// TIA Portal V18 export
FUNCTION "Function & start signal" : Void   // FC3, LAD
{ S7_Optimized_Access := 'TRUE' }
VERSION : 0.1
// stored: AutoNumber true, IsIECCheckEnabled false, SetENOAutomatically false, UDAEnableTagReadback false
   VAR_TEMP   // added for the SCL form of the ladder/FBD networks
      _w1 : Bool;
      _w2 : Bool;
      _w3 : Bool;
   END_VAR
BEGIN

REGION Network 1: Move dearing A Flowrate to Main register
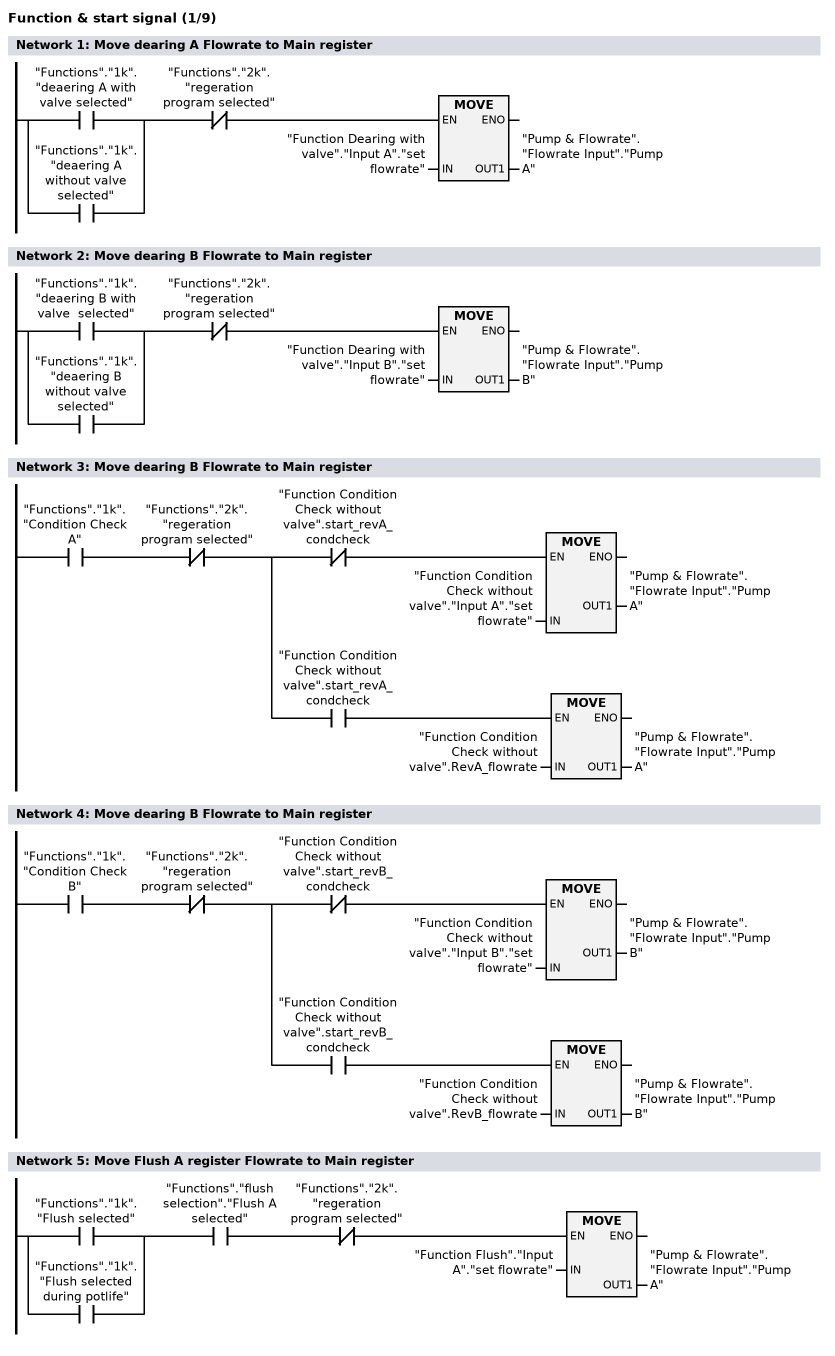
   IF ("Functions"."1k"."deaering A with valve selected" OR "Functions"."1k"."deaering A without valve selected") AND NOT "Functions"."2k"."regeration program selected" THEN
       "Pump & Flowrate"."Flowrate Input"."Pump A" := "Function Dearing with valve"."Input A"."set flowrate";
   END_IF;
END_REGION

REGION Network 2: Move dearing B Flowrate to Main register
   IF ("Functions"."1k"."deaering B with valve  selected" OR "Functions"."1k"."deaering B without valve  selected") AND NOT "Functions"."2k"."regeration program selected" THEN
       "Pump & Flowrate"."Flowrate Input"."Pump B" := "Function Dearing with valve"."Input B"."set flowrate";
   END_IF;
END_REGION

REGION Network 3: Move dearing B Flowrate to Main register
   #_w1 := "Functions"."1k"."Condition Check A" AND NOT "Functions"."2k"."regeration program selected";
   IF #_w1 AND NOT "Function ConditionCheck without valve".start_revA_condcheck THEN
       "Pump & Flowrate"."Flowrate Input"."Pump A" := "Function ConditionCheck without valve"."Input A"."set flowrate";
   END_IF;
   IF #_w1 AND "Function ConditionCheck without valve".start_revA_condcheck THEN
       "Pump & Flowrate"."Flowrate Input"."Pump A" := "Function ConditionCheck without valve".RevA_flowrate;
   END_IF;
END_REGION

REGION Network 4: Move dearing B Flowrate to Main register
   #_w1 := "Functions"."1k"."Condition Check B" AND NOT "Functions"."2k"."regeration program selected";
   IF #_w1 AND NOT "Function ConditionCheck without valve".start_revB_condcheck THEN
       "Pump & Flowrate"."Flowrate Input"."Pump B" := "Function ConditionCheck without valve"."Input B"."set flowrate";
   END_IF;
   IF #_w1 AND "Function ConditionCheck without valve".start_revB_condcheck THEN
       "Pump & Flowrate"."Flowrate Input"."Pump B" := "Function ConditionCheck without valve".RevB_flowrate;
   END_IF;
END_REGION

REGION Network 5: Move Flush A register Flowrate to Main register
   IF ("Functions"."1k"."Flush selected" OR "Functions"."1k"."Flush selected during potlife") AND "Functions"."flush selection"."Flush A selected" AND NOT "Functions"."2k"."regeration program selected" THEN
       "Pump & Flowrate"."Flowrate Input"."Pump A" := "Function Flush"."Input A"."set flowrate";
   END_IF;
END_REGION

REGION Network 6: Move Flush B register Flowrate to Main register
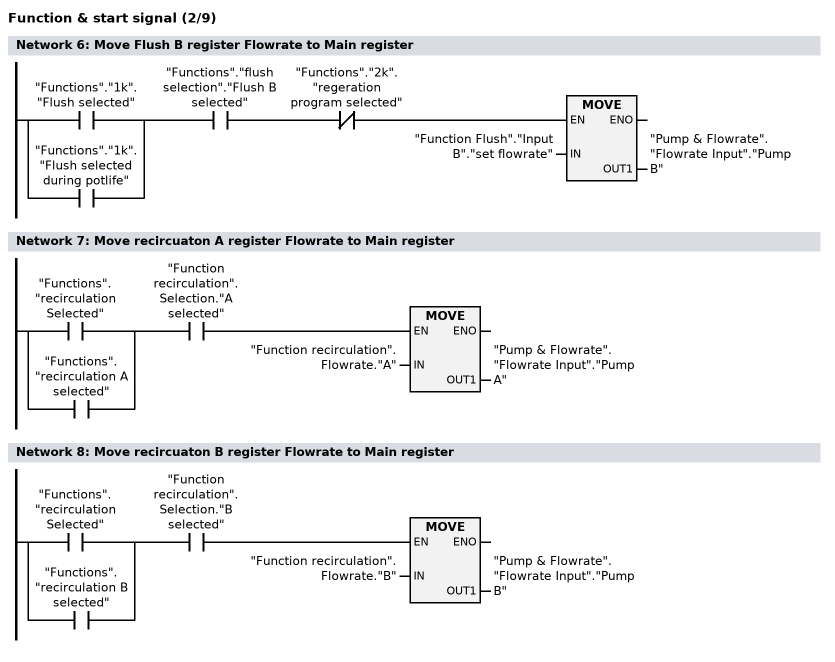
   IF ("Functions"."1k"."Flush selected" OR "Functions"."1k"."Flush selected during potlife") AND "Functions"."flush selection"."Flush B selected" AND NOT "Functions"."2k"."regeration program selected" THEN
       "Pump & Flowrate"."Flowrate Input"."Pump B" := "Function Flush"."Input B"."set flowrate";
   END_IF;
END_REGION

REGION Network 7: Move recircuaton A register Flowrate to Main register
   IF ("Functions"."recirculation Selected" OR "Functions"."recirculation A selected") AND "Function recirculation".Selection."A selected" THEN
       "Pump & Flowrate"."Flowrate Input"."Pump A" := "Function recirculation".Flowrate."A";
   END_IF;
END_REGION

REGION Network 8: Move recircuaton B register Flowrate to Main register
   IF ("Functions"."recirculation Selected" OR "Functions"."recirculation B selected") AND "Function recirculation".Selection."B selected" THEN
       "Pump & Flowrate"."Flowrate Input"."Pump B" := "Function recirculation".Flowrate."B";
   END_IF;
END_REGION

REGION Network 9: Move Metering program register Flowrate to Main register
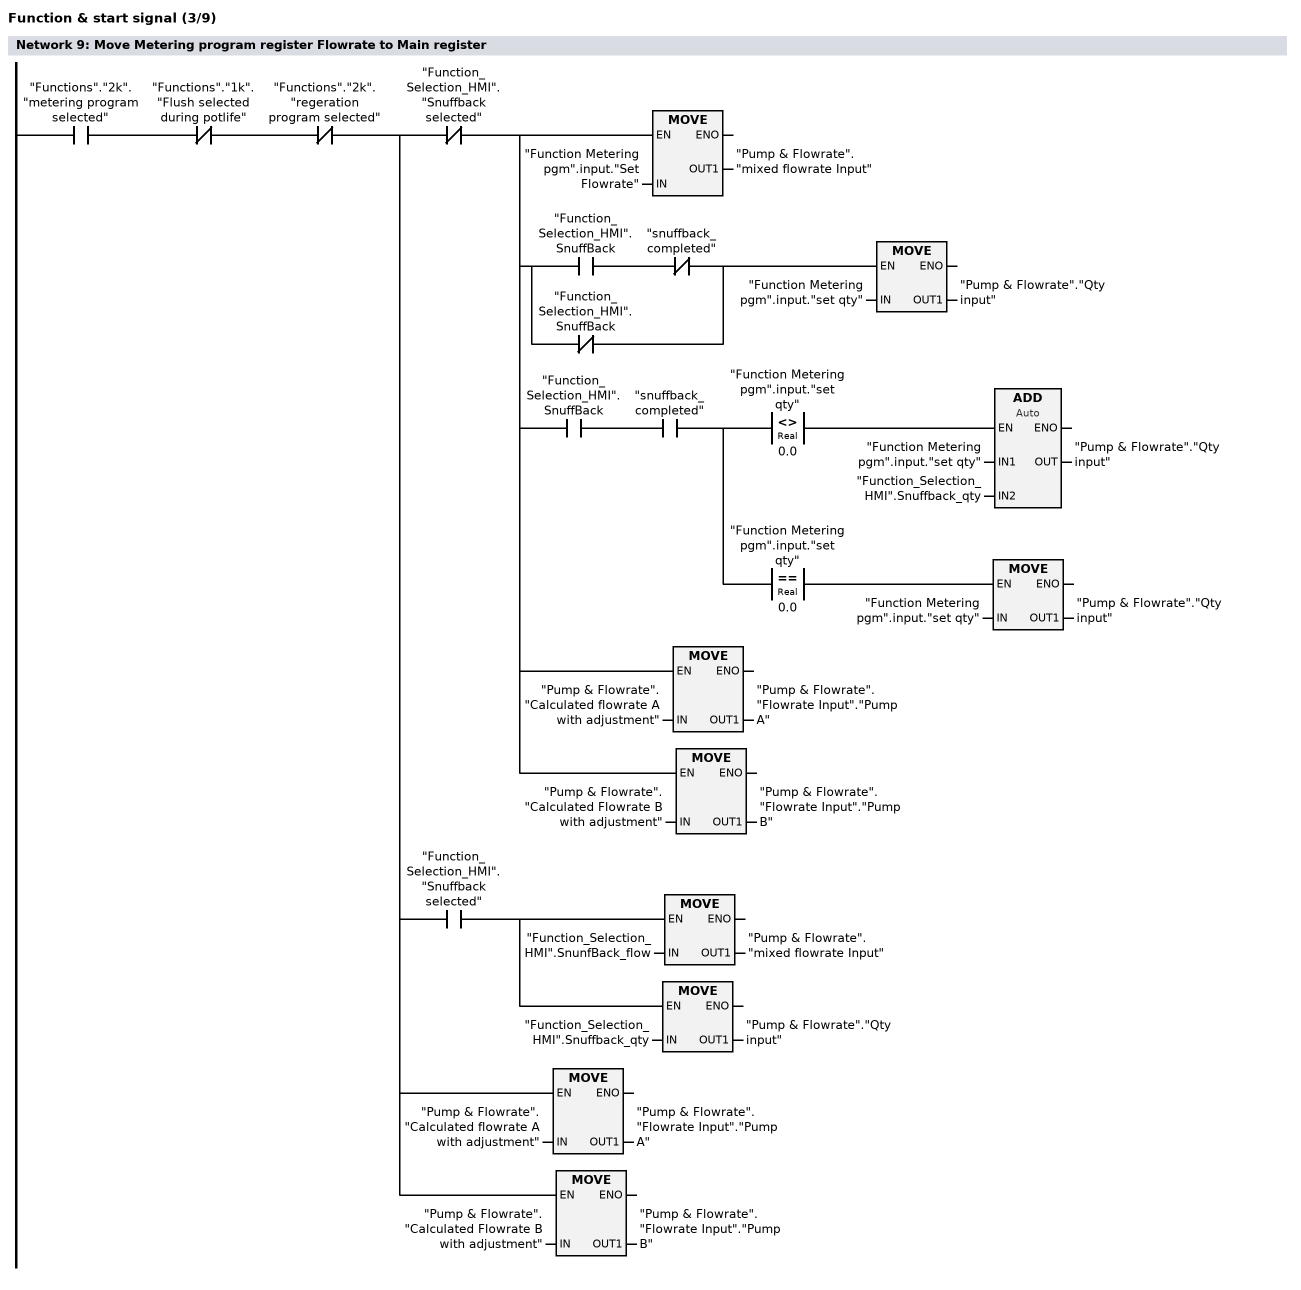
   #_w1 := "Functions"."2k"."metering program selected" AND NOT "Functions"."1k"."Flush selected during potlife" AND NOT "Functions"."2k"."regeration program selected";
   #_w2 := #_w1 AND NOT "Function_Selection_HMI"."Snuffback selected";
   IF #_w2 THEN
       "Pump & Flowrate"."mixed flowrate Input" := "Function Metering pgm".input."Set Flowrate";
   END_IF;
   IF #_w2 AND (("Function_Selection_HMI".SnuffBack AND NOT "snuffback_completed") OR NOT "Function_Selection_HMI".SnuffBack) THEN
       "Pump & Flowrate"."Qty input" := "Function Metering pgm".input."set qty";
   END_IF;
   #_w3 := #_w2 AND "Function_Selection_HMI".SnuffBack AND "snuffback_completed";
   IF #_w3 AND ("Function Metering pgm".input."set qty" <> 0.0) THEN
       "Pump & Flowrate"."Qty input" := "Function Metering pgm".input."set qty" + "Function_Selection_HMI".Snuffback_qty;
   END_IF;
   IF #_w3 AND ("Function Metering pgm".input."set qty" = 0.0) THEN
       "Pump & Flowrate"."Qty input" := "Function Metering pgm".input."set qty";
   END_IF;
   IF #_w2 THEN
       "Pump & Flowrate"."Flowrate Input"."Pump A" := "Pump & Flowrate"."Calculated flowrate A with adjustment";
       "Pump & Flowrate"."Flowrate Input"."Pump B" := "Pump & Flowrate"."Calculated Flowrate B  with adjustment";
   END_IF;
   IF #_w1 AND "Function_Selection_HMI"."Snuffback selected" THEN
       "Pump & Flowrate"."mixed flowrate Input" := "Function_Selection_HMI".SnunfBack_flow;
       "Pump & Flowrate"."Qty input" := "Function_Selection_HMI".Snuffback_qty;
   END_IF;
   IF #_w1 THEN
       "Pump & Flowrate"."Flowrate Input"."Pump A" := "Pump & Flowrate"."Calculated flowrate A with adjustment";
       "Pump & Flowrate"."Flowrate Input"."Pump B" := "Pump & Flowrate"."Calculated Flowrate B  with adjustment";
   END_IF;
END_REGION

REGION Network 10: Move shot Metering register Flowrate to Main register
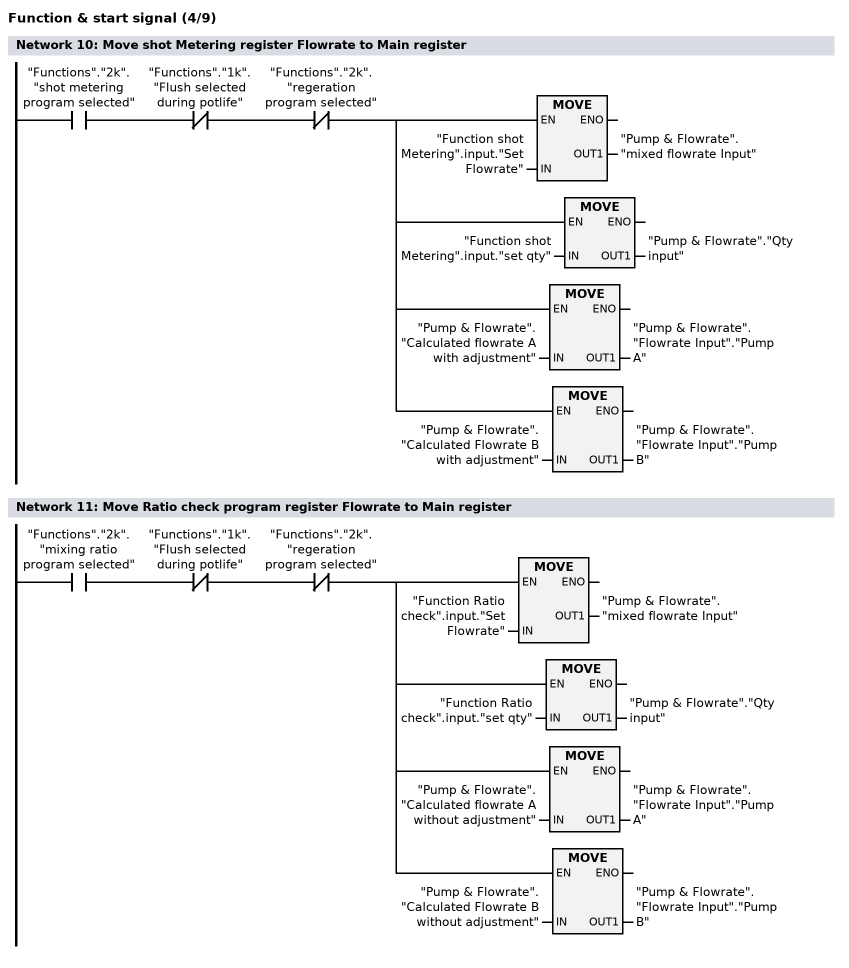
   IF "Functions"."2k"."shot metering program selected" AND NOT "Functions"."1k"."Flush selected during potlife" AND NOT "Functions"."2k"."regeration program selected" THEN
       "Pump & Flowrate"."mixed flowrate Input" := "Function shot Metering".input."Set Flowrate";
       "Pump & Flowrate"."Qty input" := "Function shot Metering".input."set qty";
       "Pump & Flowrate"."Flowrate Input"."Pump A" := "Pump & Flowrate"."Calculated flowrate A with adjustment";
       "Pump & Flowrate"."Flowrate Input"."Pump B" := "Pump & Flowrate"."Calculated Flowrate B  with adjustment";
   END_IF;
END_REGION

REGION Network 11: Move Ratio check program register Flowrate to Main register
   IF "Functions"."2k"."mixing ratio program selected" AND NOT "Functions"."1k"."Flush selected during potlife" AND NOT "Functions"."2k"."regeration program selected" THEN
       "Pump & Flowrate"."mixed flowrate Input" := "Function Ratio check".input."Set Flowrate";
       "Pump & Flowrate"."Qty input" := "Function Ratio check".input."set qty";
       "Pump & Flowrate"."Flowrate Input"."Pump A" := "Pump & Flowrate"."Calculated flowrate A without adjustment";
       "Pump & Flowrate"."Flowrate Input"."Pump B" := "Pump & Flowrate"."Calculated Flowrate B without adjustment";
   END_IF;
END_REGION

REGION Network 12: Move Pre run program register Flowrate to Main register
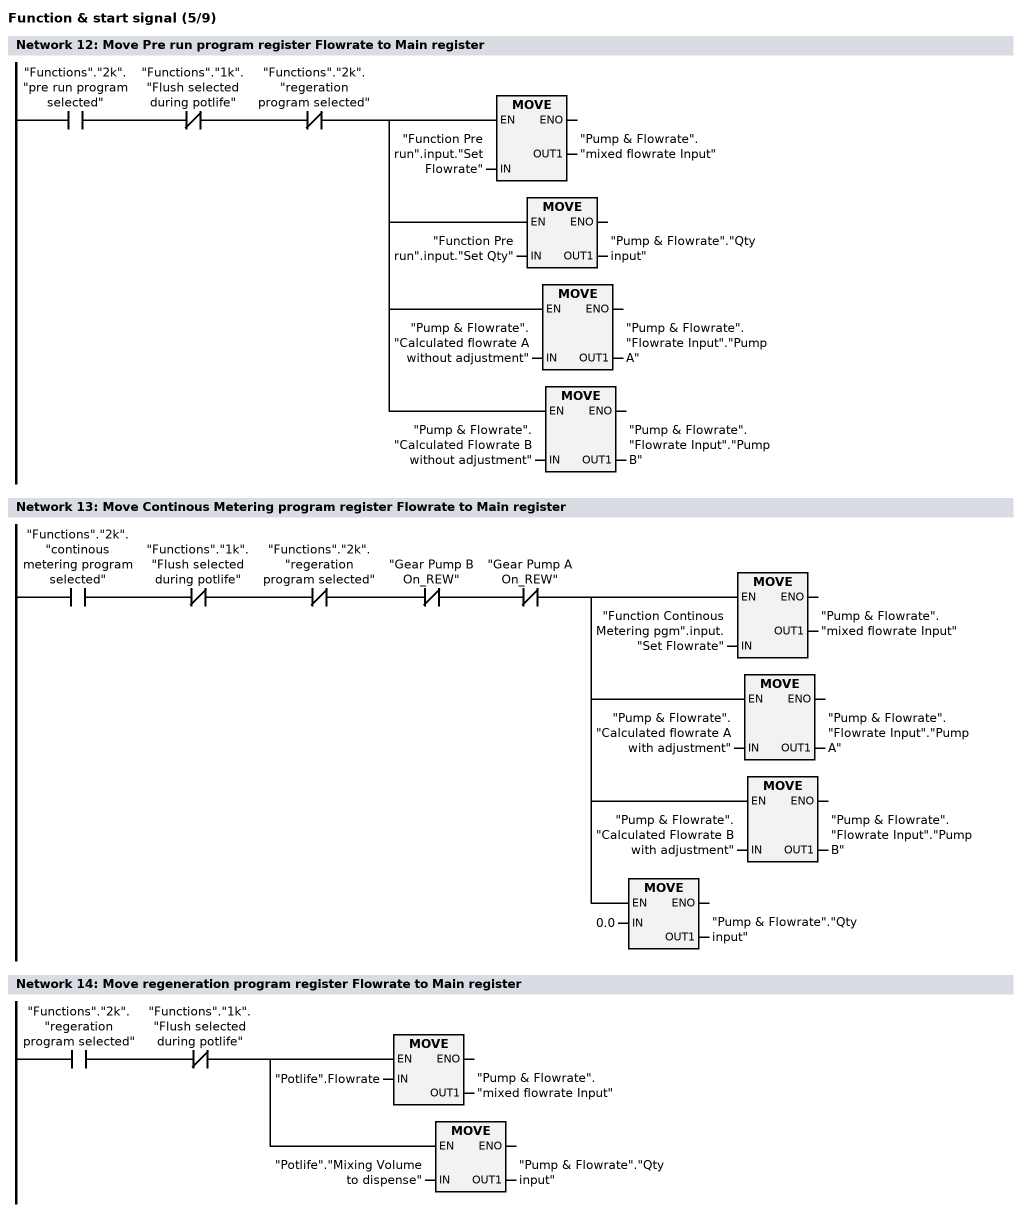
   IF "Functions"."2k"."pre run program selected" AND NOT "Functions"."1k"."Flush selected during potlife" AND NOT "Functions"."2k"."regeration program selected" THEN
       "Pump & Flowrate"."mixed flowrate Input" := "Function Pre run".input."Set Flowrate";
       "Pump & Flowrate"."Qty input" := "Function Pre run".input."Set Qty";
       "Pump & Flowrate"."Flowrate Input"."Pump A" := "Pump & Flowrate"."Calculated flowrate A without adjustment";
       "Pump & Flowrate"."Flowrate Input"."Pump B" := "Pump & Flowrate"."Calculated Flowrate B without adjustment";
   END_IF;
END_REGION

REGION Network 13: Move Continous Metering program register Flowrate to Main register
   IF "Functions"."2k"."continous metering program selected" AND NOT "Functions"."1k"."Flush selected during potlife" AND NOT "Functions"."2k"."regeration program selected" AND NOT "Gear Pump B On_REW" AND NOT "Gear Pump A On_REW" THEN
       "Pump & Flowrate"."mixed flowrate Input" := "Function Continous Metering pgm".input."Set Flowrate";
       "Pump & Flowrate"."Flowrate Input"."Pump A" := "Pump & Flowrate"."Calculated flowrate A with adjustment";
       "Pump & Flowrate"."Flowrate Input"."Pump B" := "Pump & Flowrate"."Calculated Flowrate B  with adjustment";
       "Pump & Flowrate"."Qty input" := 0.0;
   END_IF;
END_REGION

REGION Network 14: Move regeneration program register Flowrate to Main register
   IF "Functions"."2k"."regeration program selected" AND NOT "Functions"."1k"."Flush selected during potlife" THEN
       "Pump & Flowrate"."mixed flowrate Input" := "Potlife".Flowrate;
       "Pump & Flowrate"."Qty input" := "Potlife"."Mixing Volume to dispense";
   END_IF;
END_REGION

REGION Network 15: Dearing with valve A start/stop
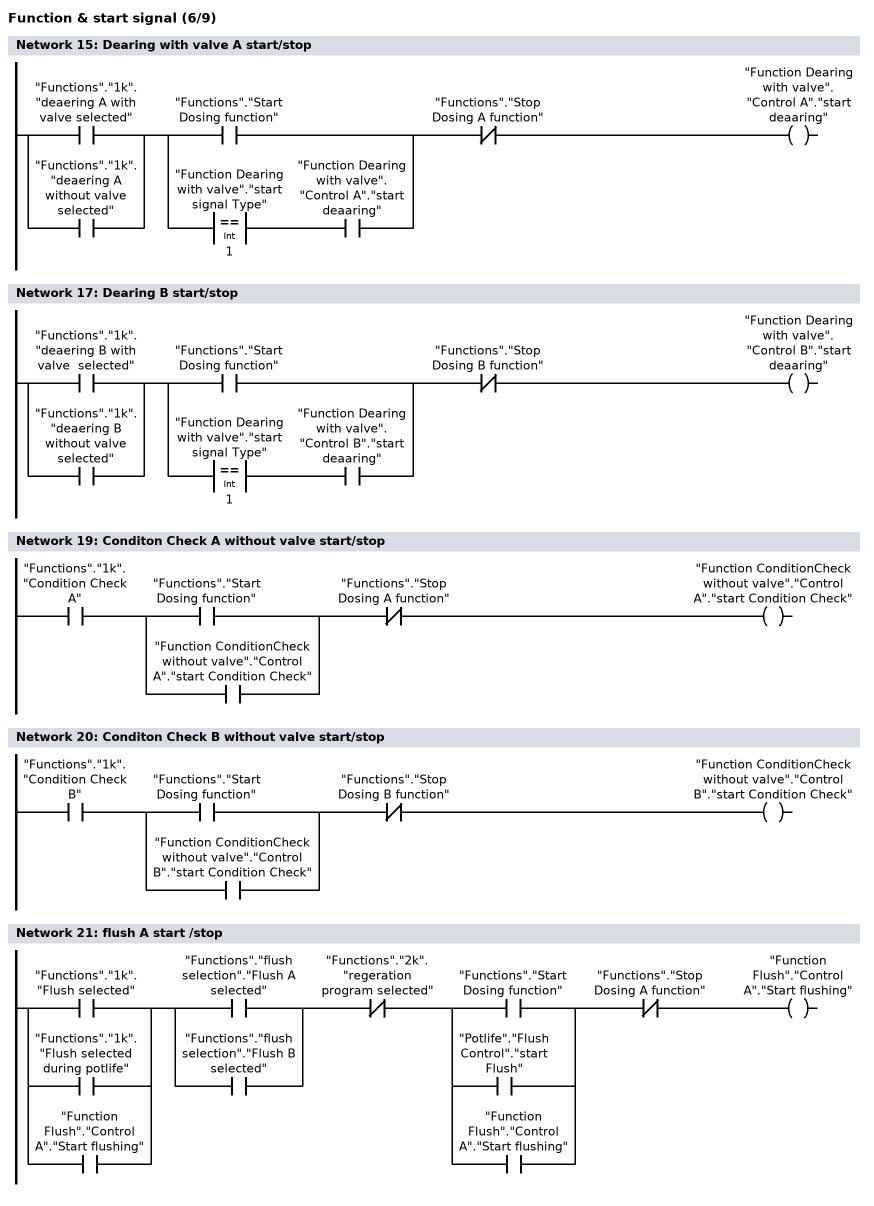
   RUNG wire#powerrail
      Contact( "Functions"."1k"."deaering A with valve selected" )
      wire#w1
      Contact( "Functions"."Start Dosing function" )
      wire#w2
      I_Contact( "Functions"."Stop Dosing A function" )
      Coil( "Function Dearing with valve"."Control A"."start deaaring" )
   END_RUNG
   RUNG wire#powerrail
      Contact( "Functions"."1k"."deaering A without valve selected" )
   END_RUNG wire#w1
   RUNG wire#w1
      { S7_Templates := "SrcType := Int" } EQ_Contact(in1 := "Function Dearing with valve"."start signal Type", in2 := 1)
      Contact( "Function Dearing with valve"."Control A"."start deaaring" )
   END_RUNG wire#w2
   // the same network as SCL:
   "Function Dearing with valve"."Control A"."start deaaring" := ("Functions"."1k"."deaering A with valve selected" OR "Functions"."1k"."deaering A without valve selected") AND ("Functions"."Start Dosing function" OR (("Function Dearing with valve"."start signal Type" = 1) AND "Function Dearing with valve"."Control A"."start deaaring")) AND NOT "Functions"."Stop Dosing A function";
END_REGION

REGION Network 16: Dearing without valve A start/stop
END_REGION

REGION Network 17: Dearing B start/stop
   RUNG wire#powerrail
      Contact( "Functions"."1k"."deaering B with valve  selected" )
      wire#w1
      Contact( "Functions"."Start Dosing function" )
      wire#w2
      I_Contact( "Functions"."Stop Dosing B function" )
      Coil( "Function Dearing with valve"."Control B"."start deaaring" )
   END_RUNG
   RUNG wire#powerrail
      Contact( "Functions"."1k"."deaering B without valve  selected" )
   END_RUNG wire#w1
   RUNG wire#w1
      { S7_Templates := "SrcType := Int" } EQ_Contact(in1 := "Function Dearing with valve"."start signal Type", in2 := 1)
      Contact( "Function Dearing with valve"."Control B"."start deaaring" )
   END_RUNG wire#w2
   // the same network as SCL:
   "Function Dearing with valve"."Control B"."start deaaring" := ("Functions"."1k"."deaering B with valve  selected" OR "Functions"."1k"."deaering B without valve  selected") AND ("Functions"."Start Dosing function" OR (("Function Dearing with valve"."start signal Type" = 1) AND "Function Dearing with valve"."Control B"."start deaaring")) AND NOT "Functions"."Stop Dosing B function";
END_REGION

REGION Network 18: Dearing B without valve start/stop
END_REGION

REGION Network 19: Conditon Check A without valve start/stop
   RUNG wire#powerrail
      Contact( "Functions"."1k"."Condition Check A" )
      wire#w1
      Contact( "Functions"."Start Dosing function" )
      wire#w2
      I_Contact( "Functions"."Stop Dosing A function" )
      Coil( "Function ConditionCheck without valve"."Control A"."start Condition Check" )
   END_RUNG
   RUNG wire#w1
      Contact( "Function ConditionCheck without valve"."Control A"."start Condition Check" )
   END_RUNG wire#w2
   // the same network as SCL:
   "Function ConditionCheck without valve"."Control A"."start Condition Check" := "Functions"."1k"."Condition Check A" AND ("Functions"."Start Dosing function" OR "Function ConditionCheck without valve"."Control A"."start Condition Check") AND NOT "Functions"."Stop Dosing A function";
END_REGION

REGION Network 20: Conditon Check B without valve start/stop
   RUNG wire#powerrail
      Contact( "Functions"."1k"."Condition Check B" )
      wire#w1
      Contact( "Functions"."Start Dosing function" )
      wire#w2
      I_Contact( "Functions"."Stop Dosing B function" )
      Coil( "Function ConditionCheck without valve"."Control B"."start Condition Check" )
   END_RUNG
   RUNG wire#w1
      Contact( "Function ConditionCheck without valve"."Control B"."start Condition Check" )
   END_RUNG wire#w2
   // the same network as SCL:
   "Function ConditionCheck without valve"."Control B"."start Condition Check" := "Functions"."1k"."Condition Check B" AND ("Functions"."Start Dosing function" OR "Function ConditionCheck without valve"."Control B"."start Condition Check") AND NOT "Functions"."Stop Dosing B function";
END_REGION

REGION Network 21: flush A start /stop
   RUNG wire#powerrail
      Contact( "Functions"."1k"."Flush selected" )
      wire#w1
      Contact( "Functions"."flush selection"."Flush A selected" )
      wire#w2
      I_Contact( "Functions"."2k"."regeration program selected" )
      wire#w3
      Contact( "Functions"."Start Dosing function" )
      wire#w4
      I_Contact( "Functions"."Stop Dosing A function" )
      Coil( "Function Flush"."Control A"."Start flushing" )
   END_RUNG
   RUNG wire#powerrail
      Contact( "Functions"."1k"."Flush selected during potlife" )
   END_RUNG wire#w1
   RUNG wire#powerrail
      Contact( "Function Flush"."Control A"."Start flushing" )
   END_RUNG wire#w1
   RUNG wire#w1
      Contact( "Functions"."flush selection"."Flush B selected" )
   END_RUNG wire#w2
   RUNG wire#w3
      Contact( "Potlife"."Flush Control"."start Flush" )
   END_RUNG wire#w4
   RUNG wire#w3
      Contact( "Function Flush"."Control A"."Start flushing" )
   END_RUNG wire#w4
   // the same network as SCL:
   "Function Flush"."Control A"."Start flushing" := ("Functions"."1k"."Flush selected" OR "Functions"."1k"."Flush selected during potlife" OR "Function Flush"."Control A"."Start flushing") AND ("Functions"."flush selection"."Flush A selected" OR "Functions"."flush selection"."Flush B selected") AND NOT "Functions"."2k"."regeration program selected" AND ("Functions"."Start Dosing function" OR "Potlife"."Flush Control"."start Flush" OR "Function Flush"."Control A"."Start flushing") AND NOT "Functions"."Stop Dosing A function";
END_REGION

REGION Network 22: flush B start /stop
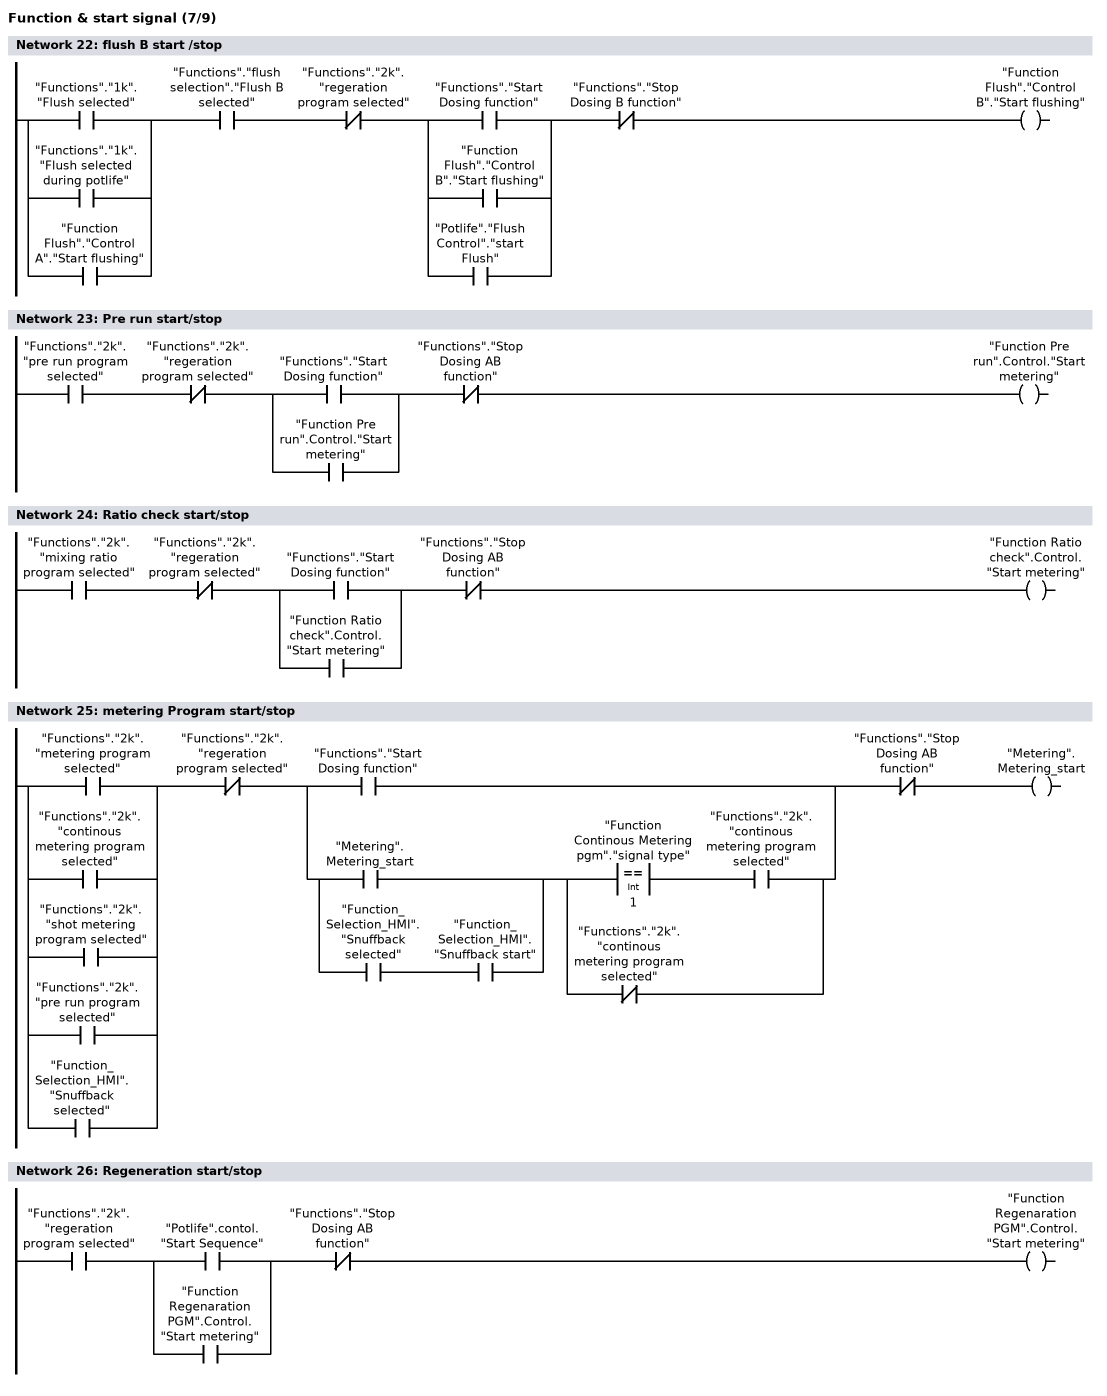
   RUNG wire#powerrail
      Contact( "Functions"."1k"."Flush selected" )
      wire#w1
      Contact( "Functions"."flush selection"."Flush B selected" )
      I_Contact( "Functions"."2k"."regeration program selected" )
      wire#w2
      Contact( "Functions"."Start Dosing function" )
      wire#w3
      I_Contact( "Functions"."Stop Dosing B function" )
      Coil( "Function Flush"."Control B"."Start flushing" )
   END_RUNG
   RUNG wire#powerrail
      Contact( "Functions"."1k"."Flush selected during potlife" )
   END_RUNG wire#w1
   RUNG wire#powerrail
      Contact( "Function Flush"."Control A"."Start flushing" )
   END_RUNG wire#w1
   RUNG wire#w2
      Contact( "Function Flush"."Control B"."Start flushing" )
   END_RUNG wire#w3
   RUNG wire#w2
      Contact( "Potlife"."Flush Control"."start Flush" )
   END_RUNG wire#w3
   // the same network as SCL:
   "Function Flush"."Control B"."Start flushing" := ("Functions"."1k"."Flush selected" OR "Functions"."1k"."Flush selected during potlife" OR "Function Flush"."Control A"."Start flushing") AND "Functions"."flush selection"."Flush B selected" AND NOT "Functions"."2k"."regeration program selected" AND ("Functions"."Start Dosing function" OR "Function Flush"."Control B"."Start flushing" OR "Potlife"."Flush Control"."start Flush") AND NOT "Functions"."Stop Dosing B function";
END_REGION

REGION Network 23: Pre run start/stop
   RUNG wire#powerrail
      Contact( "Functions"."2k"."pre run program selected" )
      I_Contact( "Functions"."2k"."regeration program selected" )
      wire#w1
      Contact( "Functions"."Start Dosing function" )
      wire#w2
      I_Contact( "Functions"."Stop Dosing AB function" )
      Coil( "Function Pre run".Control."Start metering" )
   END_RUNG
   RUNG wire#w1
      Contact( "Function Pre run".Control."Start metering" )
   END_RUNG wire#w2
   // the same network as SCL:
   "Function Pre run".Control."Start metering" := "Functions"."2k"."pre run program selected" AND NOT "Functions"."2k"."regeration program selected" AND ("Functions"."Start Dosing function" OR "Function Pre run".Control."Start metering") AND NOT "Functions"."Stop Dosing AB function";
END_REGION

REGION Network 24: Ratio check start/stop
   RUNG wire#powerrail
      Contact( "Functions"."2k"."mixing ratio program selected" )
      I_Contact( "Functions"."2k"."regeration program selected" )
      wire#w1
      Contact( "Functions"."Start Dosing function" )
      wire#w2
      I_Contact( "Functions"."Stop Dosing AB function" )
      Coil( "Function Ratio check".Control."Start metering" )
   END_RUNG
   RUNG wire#w1
      Contact( "Function Ratio check".Control."Start metering" )
   END_RUNG wire#w2
   // the same network as SCL:
   "Function Ratio check".Control."Start metering" := "Functions"."2k"."mixing ratio program selected" AND NOT "Functions"."2k"."regeration program selected" AND ("Functions"."Start Dosing function" OR "Function Ratio check".Control."Start metering") AND NOT "Functions"."Stop Dosing AB function";
END_REGION

REGION Network 25: metering Program start/stop
   RUNG wire#powerrail
      Contact( "Functions"."2k"."metering program selected" )
      wire#w1
      I_Contact( "Functions"."2k"."regeration program selected" )
      wire#w2
      Contact( "Functions"."Start Dosing function" )
      wire#w3
      I_Contact( "Functions"."Stop Dosing AB function" )
      Coil( "Metering".Metering_start )
   END_RUNG
   RUNG wire#powerrail
      Contact( "Functions"."2k"."continous metering program selected" )
   END_RUNG wire#w1
   RUNG wire#powerrail
      Contact( "Functions"."2k"."shot metering program selected" )
   END_RUNG wire#w1
   RUNG wire#powerrail
      Contact( "Functions"."2k"."pre run program selected" )
   END_RUNG wire#w1
   RUNG wire#powerrail
      Contact( "Function_Selection_HMI"."Snuffback selected" )
   END_RUNG wire#w1
   RUNG wire#w2
      Contact( "Metering".Metering_start )
      wire#w4
      { S7_Templates := "SrcType := Int" } EQ_Contact(in1 := "Function Continous Metering pgm"."signal type", in2 := 1)
      Contact( "Functions"."2k"."continous metering program selected" )
   END_RUNG wire#w3
   RUNG wire#w2
      Contact( "Function_Selection_HMI"."Snuffback selected" )
      Contact( "Function_Selection_HMI"."Snuffback start" )
   END_RUNG wire#w4
   RUNG wire#w4
      I_Contact( "Functions"."2k"."continous metering program selected" )
   END_RUNG wire#w3
   // the same network as SCL:
   "Metering".Metering_start := ("Functions"."2k"."metering program selected" OR "Functions"."2k"."continous metering program selected" OR "Functions"."2k"."shot metering program selected" OR "Functions"."2k"."pre run program selected" OR "Function_Selection_HMI"."Snuffback selected") AND NOT "Functions"."2k"."regeration program selected" AND ("Functions"."Start Dosing function" OR (("Metering".Metering_start OR ("Function_Selection_HMI"."Snuffback selected" AND "Function_Selection_HMI"."Snuffback start")) AND ((("Function Continous Metering pgm"."signal type" = 1) AND "Functions"."2k"."continous metering program selected") OR NOT "Functions"."2k"."continous metering program selected"))) AND NOT "Functions"."Stop Dosing AB function";
END_REGION

REGION Network 26: Regeneration start/stop
   RUNG wire#powerrail
      Contact( "Functions"."2k"."regeration program selected" )
      wire#w1
      Contact( "Potlife".contol."Start Sequence" )
      wire#w2
      I_Contact( "Functions"."Stop Dosing AB function" )
      Coil( "Function Regenaration PGM".Control."Start metering" )
   END_RUNG
   RUNG wire#w1
      Contact( "Function Regenaration PGM".Control."Start metering" )
   END_RUNG wire#w2
   // the same network as SCL:
   "Function Regenaration PGM".Control."Start metering" := "Functions"."2k"."regeration program selected" AND ("Potlife".contol."Start Sequence" OR "Function Regenaration PGM".Control."Start metering") AND NOT "Functions"."Stop Dosing AB function";
END_REGION

REGION Network 27: metering Shot start/stop
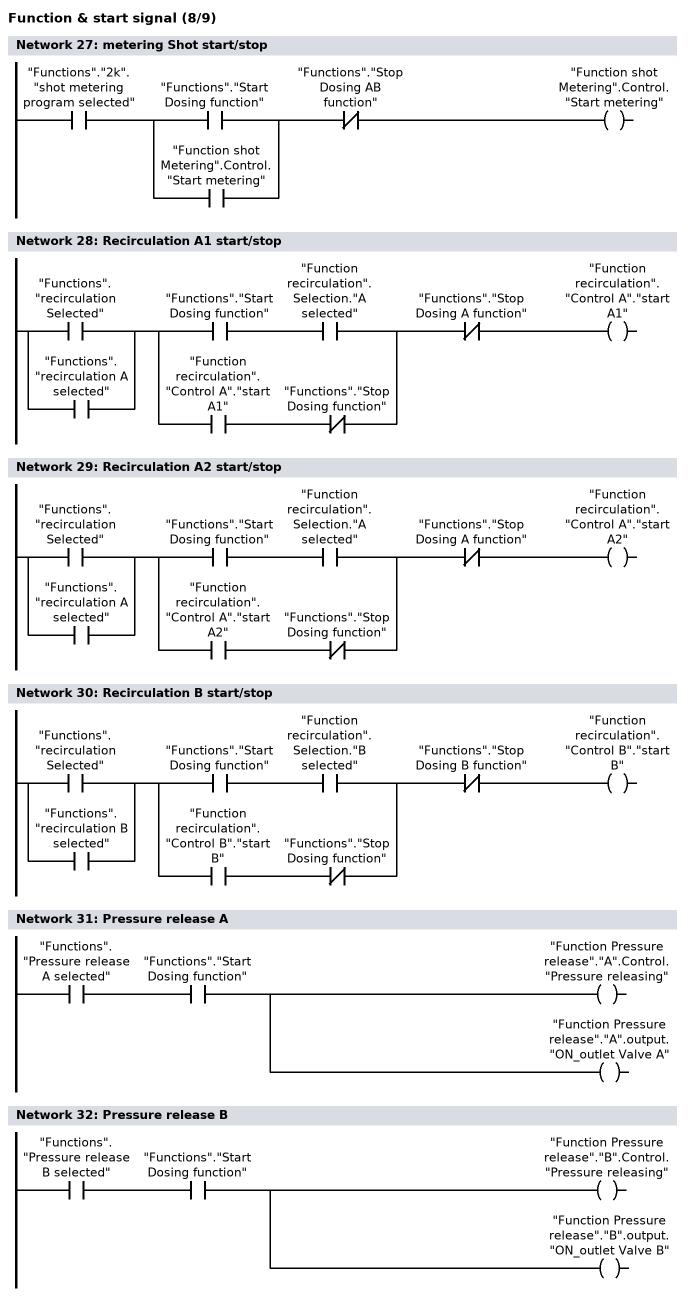
   RUNG wire#powerrail
      Contact( "Functions"."2k"."shot metering program selected" )
      wire#w1
      Contact( "Functions"."Start Dosing function" )
      wire#w2
      I_Contact( "Functions"."Stop Dosing AB function" )
      Coil( "Function shot Metering".Control."Start metering" )
   END_RUNG
   RUNG wire#w1
      Contact( "Function shot Metering".Control."Start metering" )
   END_RUNG wire#w2
   // the same network as SCL:
   "Function shot Metering".Control."Start metering" := "Functions"."2k"."shot metering program selected" AND ("Functions"."Start Dosing function" OR "Function shot Metering".Control."Start metering") AND NOT "Functions"."Stop Dosing AB function";
END_REGION

REGION Network 28: Recirculation A1 start/stop
   RUNG wire#powerrail
      Contact( "Functions"."recirculation Selected" )
      wire#w1
      Contact( "Functions"."Start Dosing function" )
      Contact( "Function recirculation".Selection."A selected" )
      wire#w2
      I_Contact( "Functions"."Stop Dosing A function" )
      Coil( "Function recirculation"."Control A"."start A1" )
   END_RUNG
   RUNG wire#powerrail
      Contact( "Functions"."recirculation A selected" )
   END_RUNG wire#w1
   RUNG wire#w1
      Contact( "Function recirculation"."Control A"."start A1" )
      I_Contact( "Functions"."Stop Dosing function" )
   END_RUNG wire#w2
   // the same network as SCL:
   "Function recirculation"."Control A"."start A1" := ("Functions"."recirculation Selected" OR "Functions"."recirculation A selected") AND (("Functions"."Start Dosing function" AND "Function recirculation".Selection."A selected") OR ("Function recirculation"."Control A"."start A1" AND NOT "Functions"."Stop Dosing function")) AND NOT "Functions"."Stop Dosing A function";
END_REGION

REGION Network 29: Recirculation A2 start/stop
   RUNG wire#powerrail
      Contact( "Functions"."recirculation Selected" )
      wire#w1
      Contact( "Functions"."Start Dosing function" )
      Contact( "Function recirculation".Selection."A selected" )
      wire#w2
      I_Contact( "Functions"."Stop Dosing A function" )
      Coil( "Function recirculation"."Control A"."start A2" )
   END_RUNG
   RUNG wire#powerrail
      Contact( "Functions"."recirculation A selected" )
   END_RUNG wire#w1
   RUNG wire#w1
      Contact( "Function recirculation"."Control A"."start A2" )
      I_Contact( "Functions"."Stop Dosing function" )
   END_RUNG wire#w2
   // the same network as SCL:
   "Function recirculation"."Control A"."start A2" := ("Functions"."recirculation Selected" OR "Functions"."recirculation A selected") AND (("Functions"."Start Dosing function" AND "Function recirculation".Selection."A selected") OR ("Function recirculation"."Control A"."start A2" AND NOT "Functions"."Stop Dosing function")) AND NOT "Functions"."Stop Dosing A function";
END_REGION

REGION Network 30: Recirculation B start/stop
   RUNG wire#powerrail
      Contact( "Functions"."recirculation Selected" )
      wire#w1
      Contact( "Functions"."Start Dosing function" )
      Contact( "Function recirculation".Selection."B selected" )
      wire#w2
      I_Contact( "Functions"."Stop Dosing B function" )
      Coil( "Function recirculation"."Control B"."start B" )
   END_RUNG
   RUNG wire#powerrail
      Contact( "Functions"."recirculation B selected" )
   END_RUNG wire#w1
   RUNG wire#w1
      Contact( "Function recirculation"."Control B"."start B" )
      I_Contact( "Functions"."Stop Dosing function" )
   END_RUNG wire#w2
   // the same network as SCL:
   "Function recirculation"."Control B"."start B" := ("Functions"."recirculation Selected" OR "Functions"."recirculation B selected") AND (("Functions"."Start Dosing function" AND "Function recirculation".Selection."B selected") OR ("Function recirculation"."Control B"."start B" AND NOT "Functions"."Stop Dosing function")) AND NOT "Functions"."Stop Dosing B function";
END_REGION

REGION Network 31: Pressure release A
   RUNG wire#powerrail
      Contact( "Functions"."Pressure release A selected" )
      Contact( "Functions"."Start Dosing function" )
      wire#w1
      Coil( "Function Pressure release"."A".Control."Pressure releasing" )
   END_RUNG
   RUNG wire#w1
      Coil( "Function Pressure release"."A".output."ON_outlet Valve A" )
   END_RUNG
   // the same network as SCL:
   "Function Pressure release"."A".Control."Pressure releasing" := "Functions"."Pressure release A selected" AND "Functions"."Start Dosing function";
   "Function Pressure release"."A".output."ON_outlet Valve A" := "Function Pressure release"."A".Control."Pressure releasing";
END_REGION

REGION Network 32: Pressure release B
   RUNG wire#powerrail
      Contact( "Functions"."Pressure release B selected" )
      Contact( "Functions"."Start Dosing function" )
      wire#w1
      Coil( "Function Pressure release"."B".Control."Pressure releasing" )
   END_RUNG
   RUNG wire#w1
      Coil( "Function Pressure release"."B".output."ON_outlet Valve B" )
   END_RUNG
   // the same network as SCL:
   "Function Pressure release"."B".Control."Pressure releasing" := "Functions"."Pressure release B selected" AND "Functions"."Start Dosing function";
   "Function Pressure release"."B".output."ON_outlet Valve B" := "Function Pressure release"."B".Control."Pressure releasing";
END_REGION

REGION Network 33: Pressure release AB
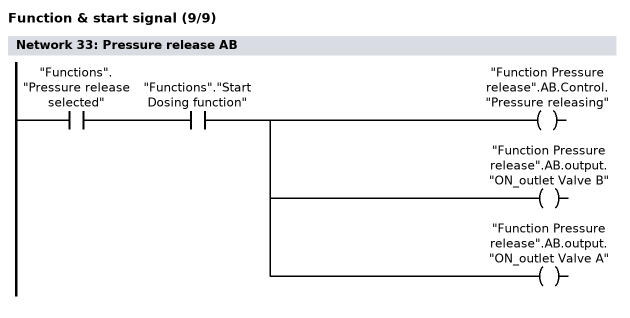
   RUNG wire#powerrail
      Contact( "Functions"."Pressure release selected" )
      Contact( "Functions"."Start Dosing function" )
      wire#w1
      Coil( "Function Pressure release".AB.Control."Pressure releasing" )
   END_RUNG
   RUNG wire#w1
      Coil( "Function Pressure release".AB.output."ON_outlet Valve B" )
   END_RUNG
   RUNG wire#w1
      Coil( "Function Pressure release".AB.output."ON_outlet Valve A" )
   END_RUNG
   // the same network as SCL:
   "Function Pressure release".AB.Control."Pressure releasing" := "Functions"."Pressure release selected" AND "Functions"."Start Dosing function";
   "Function Pressure release".AB.output."ON_outlet Valve B" := "Function Pressure release".AB.Control."Pressure releasing";
   "Function Pressure release".AB.output."ON_outlet Valve A" := "Function Pressure release".AB.Control."Pressure releasing";
END_REGION
END_FUNCTION
